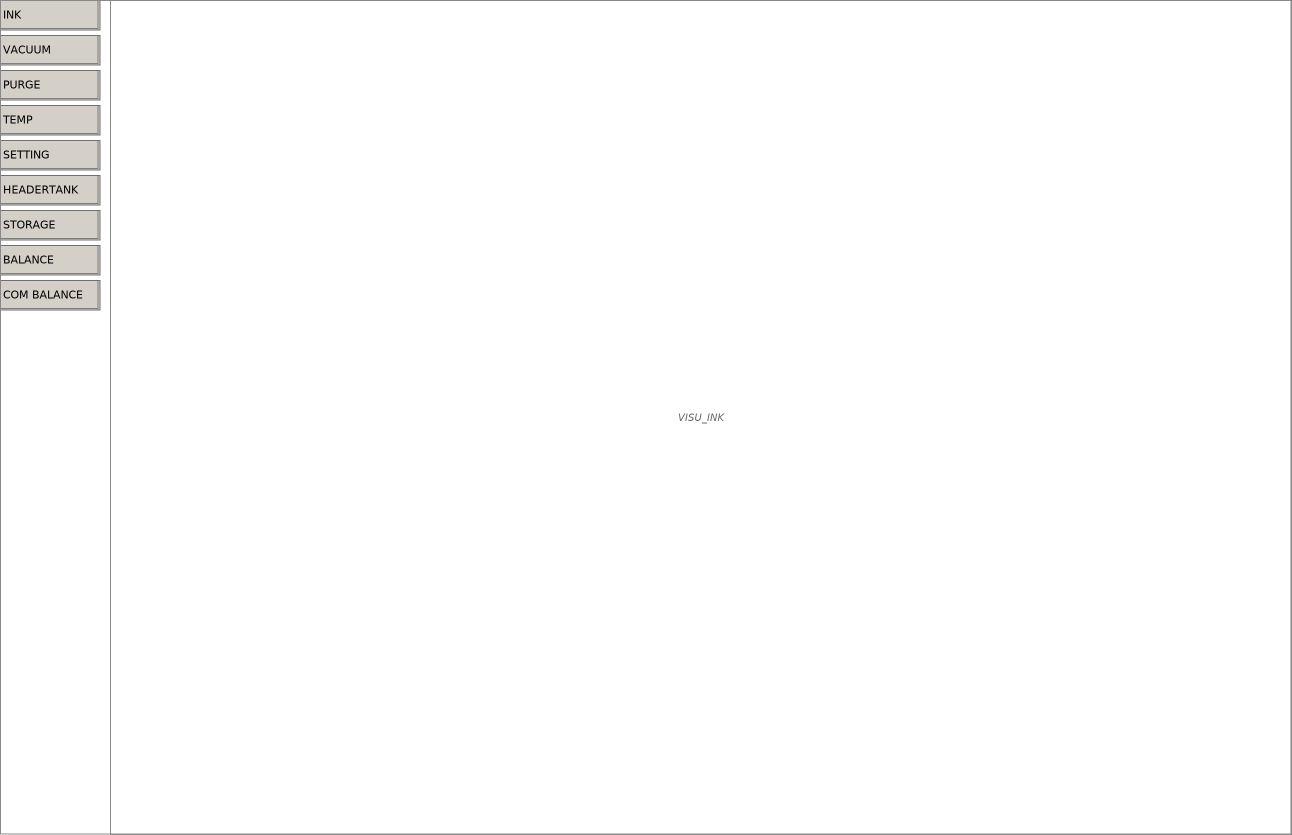
VISUALIZATION VISU_INKSYSTEM  // 1292x835
    Frame (110,0 1182x835), frame switch variable: PRG_INK.aVisuInkSystemFrameIndex
        shows VISU_INK()
        shows VISU_VACUUM()
        shows VISU_PURGE()
        shows VISU_TEMPERATUR()
        shows VISU_SETTINGS()
        shows VISU_HEADERTANK()
        shows VISU_ADS_INKSTORAGE_TANK_DVT()
        shows VISU_BALANCE()
        shows VISU_COMM_BALANCE()
    Button (0,0 100x30), "INK", colour toggle: PRG_INK.aVisuInkSystemFrameIndex = 0
        OnMouseClick: execute { PRG_INK.aVisuInkSystemFrameIndex := 0; }
    Button (0,70 100x30), "PURGE", colour toggle: PRG_INK.aVisuInkSystemFrameIndex = 2
        OnMouseClick: execute { PRG_INK.aVisuInkSystemFrameIndex := 2; }
    Button (0,105 100x30), "TEMP", colour toggle: PRG_INK.aVisuInkSystemFrameIndex = 3
        OnMouseClick: execute { PRG_INK.aVisuInkSystemFrameIndex := 3; }
    Button (0,140 100x30), "SETTING", colour toggle: PRG_INK.aVisuInkSystemFrameIndex = 4
        OnMouseClick: execute { PRG_INK.aVisuInkSystemFrameIndex := 4; }
    Button (0,210 100x30), "STORAGE", colour toggle: PRG_INK.aVisuInkSystemFrameIndex = 6
        OnMouseClick: execute { PRG_INK.aVisuInkSystemFrameIndex := 6; }
    Button (0,35 100x30), "VACUUM", colour toggle: PRG_INK.aVisuInkSystemFrameIndex = 1
        OnMouseClick: execute { PRG_INK.aVisuInkSystemFrameIndex := 1; }
    Button (0,175 100x30), "HEADERTANK", colour toggle: PRG_INK.aVisuInkSystemFrameIndex = 5
        OnMouseClick: execute { PRG_INK.aVisuInkSystemFrameIndex := 5; }
    Button (0,245 100x30), "BALANCE", colour toggle: PRG_INK.aVisuInkSystemFrameIndex = 7
        OnMouseClick: execute { PRG_INK.aVisuInkSystemFrameIndex := 7; }
    Button (0,280 100x30), "COM BALANCE", colour toggle: PRG_INK.aVisuInkSystemFrameIndex = 8
        OnMouseClick: execute { PRG_INK.aVisuInkSystemFrameIndex := 8; }
END_VISUALIZATION

(* stored: Version 1.1.0.1, ProductVersion 3.1.4024.11
   Visu VISU_INKSYSTEM: Id {1b288260-0665-4e34-aa6a-561a0c15d599} *)
